FUNCTION_BLOCK OutputAts400 EXTENDS TcoCore.TcoState IMPLEMENTS IOutputAts400
VAR_OUTPUT
    output : ARRAY[1..12] OF BOOl;
END_VAR
VAR
    selectProgramTask : SelectProgramTask(THIS^);
END_VAR

METHOD AbortTest
VAR_INPUT
    enable : BOOL;
END_VAR
THIS^.output[2] := enable;
END_METHOD

METHOD SelectProgramm : TcoCore.ITcoTaskStatus
VAR_INPUT
    programm : UINT;
END_VAR
//mind 18ms muss Select gesetzt sein

SelectProgramm := selectProgramTask.Invoke();
selectProgramTask(selectedProgram := programm, output => output);
END_METHOD

METHOD SetDummyReady
VAR_INPUT
    enable : BOOL;
END_VAR
output[5] := enable;
END_METHOD

METHOD SetManualFail
VAR_INPUT
    enable : BOOL;
END_VAR
output[4] := enable;
END_METHOD

METHOD SetManualPass
VAR_INPUT
    enable : BOOL;
END_VAR
output[3] := enable;
END_METHOD

METHOD Start
VAR_INPUT
    enable : BOOL;
END_VAR
this^.output[1] := enable;
END_METHOD

END_FUNCTION_BLOCK

(* stored: Version 1.1.0.1, ProductVersion 3.1.4024.12
   POU OutputAts400: Id {bd7aa8b3-01d0-4f2a-b42e-da0cb9424db6}, SpecialFunc None
   Method AbortTest: Id {e0d45663-ed6c-41a9-b491-4d68a84754c0}
   Method SelectProgramm: Id {94f3e723-9abd-49b8-8079-3bf1f7bee9e2}
   Method SetDummyReady: Id {290d1db9-9de7-4da1-be79-3003f6c53c37}
   Method SetManualFail: Id {1b6deb94-7eed-490a-b11a-5717d5885917}
   Method SetManualPass: Id {ac847f6f-4cd5-46cc-9b3e-25d42092aa04}
   Method Start: Id {ffe48cac-4552-44f6-bb74-95127658e21f} *)
